{attribute 'reflection'}
FUNCTION_BLOCK PUBLIC ABSTRACT FB_LogHandlerBase // Base class for all log handlers
VAR_OUTPUT
	{attribute 'instance-path'} 
    {attribute 'noinit'}
	sInstancePath : STRING; // Instance path of the function block
END_VAR

METHOD INTERNAL ABSTRACT M_AddToLog
VAR_INPUT
	sMsg : T_MaxString; // The message to be logged
	eLevel : E_LogLevel; // Log level (debug, info, warn, etc.)
END_VAR
END_METHOD

END_FUNCTION_BLOCK

(* stored: Version 1.1.0.1, ProductVersion 3.1.4024.11
   POU FB_LogHandlerBase: Id {c49e850d-7280-093e-30c8-6ebb7bc3ee12}, SpecialFunc None
   Method M_AddToLog: Id {ebb0fcf3-f03d-0288-2f6b-00eb9ae0a605} *)
